Fanuc KAREL source: mth_sin.kl

PROGRAM mth_sin
%NOBUSYLAMP
%NOLOCKGROUP

VAR
	out_reg : INTEGER
	angle : REAL
%from tpe.klh %import get_real_arg,get_int_arg
%from registers.klh %import set_real
%from math.builtins.klh %import sin

BEGIN
	angle = tpe__get_real_arg(1)
	out_reg = tpe__get_int_arg(2)
	registers__set_real(out_reg, math__sin(angle))
END mth_sin
